FUNCTION_BLOCK EC_Piston (* Commands of Piston as output values, in timed phases: Stop=0, Up=1, Down=2 *)
  (* Standard: 61499-2 *)
  (* Version 0.1, 2026-09-28, Project contributors, AAU Smart Production Lab *)
  PACKAGE stoppering;
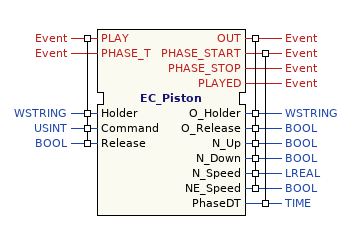
  EVENT_INPUT
    PLAY WITH Holder, Command, Release;
    PHASE_T;
  END_EVENT
  EVENT_OUTPUT
    OUT WITH O_Holder, O_Release, N_Up, N_Down, N_Speed, NE_Speed;
    PHASE_START WITH PhaseDT;
    PHASE_STOP;
    PLAYED;
  END_EVENT
  VAR_INPUT
    Holder : WSTRING;
    Command : USINT;
    Release : BOOL;
  END_VAR
  VAR_OUTPUT
    O_Holder : WSTRING;
    O_Release : BOOL;
    N_Up : BOOL;
    N_Down : BOOL;
    N_Speed : LREAL;
    NE_Speed : BOOL;
    PhaseDT : TIME;
  END_VAR
  VAR
    Phase : USINT;
    Timed : BOOL;
  END_VAR
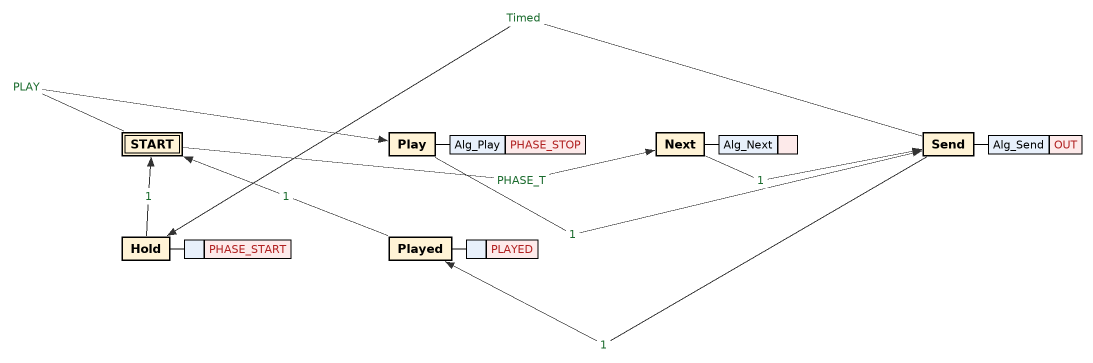
  EC_STATES
    START;
    Play : Alg_Play -> PHASE_STOP;
    Next : Alg_Next;
    Send : Alg_Send -> OUT;
    Hold : -> PHASE_START;
    Played : -> PLAYED;
  END_STATES
  EC_TRANSITIONS
    START TO Play := PLAY;
    START TO Next := PHASE_T;
    Play TO Send := 1;
    Next TO Send := 1;
    Send TO Hold := Timed;
    Send TO Played := 1;
    Hold TO START := 1;
    Played TO START := 1;
  END_TRANSITIONS
  ALGORITHM Alg_Play IN ST:
Phase := 0;
  END_ALGORITHM
  ALGORITHM Alg_Next IN ST:
Phase := Phase + 1;
  END_ALGORITHM
  ALGORITHM Alg_Send IN ST:
N_Up := FALSE;
N_Down := FALSE;
N_Speed := 0.0;
NE_Speed := FALSE;
Timed := FALSE;
PhaseDT := T#0ms;
IF Command = 1 THEN
  N_Up := TRUE;
  N_Speed := 200.0;
  NE_Speed := TRUE;
ELSIF Command = 2 THEN
  N_Down := TRUE;
  N_Speed := 200.0;
  NE_Speed := TRUE;
END_IF;
O_Holder := Holder;
O_Release := Release AND NOT Timed;
  END_ALGORITHM
END_FUNCTION_BLOCK
